// TIA Portal V19 export
DATA_BLOCK "A0302_PareggiatoreCoda_PERS"   // DB120
// stored: MemoryReserve 100
   VAR RETAIN
      Par : Struct
         Ax { S7_SetPoint := 'True'} : "Positioning_DOL_Machine_Par";
         Ax_Pers { ExternalAccessible := 'False'; ExternalVisible := 'False'; ExternalWritable := 'False'} : "Positioning_DOL_Machine_Pers_Data";
         Enc : "PosFbk_RTN";
         Ax_Aut { S7_SetPoint := 'True'} : "A0301_Mach_Speed_Par";
         Bloccaggio_Sens : Struct
            "2191B1" : "Analogic_SensorManagement_Par";
            SogliaWork { S7_SetPoint := 'True'} : Real := 0.0;
         END_STRUCT;
         CarroPareggCoda : Struct
            Delay_StartMove : Time := T#100MS;
            Preset { S7_SetPoint := 'True'} : LReal := 477.68;
         END_STRUCT;
         Cremaliera : Struct
            Modulo { S7_SetPoint := 'True'} : LReal := 2.5;
            Passo { S7_SetPoint := 'True'} : LReal := 7.854;
         END_STRUCT;
      END_STRUCT;
      Par_Sens : Struct
         AI { S7_SetPoint := 'True'} : "Analogic_SensorManagement_Par";
      END_STRUCT;
      Data_Sens { S7_SetPoint := 'True'} : "Analogic_SensorManagement_Data";
      Par_MachSens { S7_SetPoint := 'True'} : "A0301_Mach_Sens_Par";
      IEC_SP : Struct
         FTC_Input : Struct
            TON_PT : Time := T#10MS;
            TOF_PT : Time := T#100MS;
         END_STRUCT;
         FTC_Output : Struct
            TON_PT : Time := T#10MS;
            TOF_PT : Time := T#10MS;
         END_STRUCT;
         FTC_PresentMat : Struct
            TON_PT : Time := T#500MS;
            TOF_PT : Time := T#500MS;
         END_STRUCT;
         Check_2119B1 { ExternalAccessible := 'False'; ExternalVisible := 'False'; ExternalWritable := 'False'} : Struct
            TON_PT : Time := T#500MS;
         END_STRUCT;
      END_STRUCT;
   END_VAR
BEGIN
   Par.Ax.PosTolerance := 1.0;
   Par.Ax.Minus_Limit := 457.6;
   Par.Ax.Plus_Limit := 2845.0;
   Par.Ax.PreCutOff := 0.2;
   Par.Ax.PreEndLowSpeed := 2.0;
   Par.Ax.PreEndMedSpeed := 5.0;
   Par.Ax.LowSpeed := 2.0;
   Par.Ax.MedSpeed := 5.0;
   Par.Ax.HighSpeed := 50.0;
   Par.Ax.Man_Speed := 50.0;
   Par.Ax_Pers.AxisHomed := TRUE;
   Par.Enc.Preset.Pulses := 1_666_530_232;
   Par.Enc.Preset.Units := 477.68;
   Par.Enc.Config.Resolution := 125.663706143592;
   Par.Ax_Aut.SemiAut_Vel := 50.0;
   Par.Ax_Aut.Aut_Vel := 50.0;
   Par.Ax_Aut.Aut_Acc := 1.0;
   Par.Ax_Aut.Aut_Dec := 1.0;
   Par.Bloccaggio_Sens."2191B1".Enable := TRUE;
   Par.Bloccaggio_Sens."2191B1".RangeLow := 0.0;
   Par.Bloccaggio_Sens."2191B1".RangeHigh := 0.0;
   Par_Sens.AI.Enable := TRUE;
   Par_Sens.AI.RangeLow := 43.0;
   Par_Sens.AI.RangeHigh := 133.7;
   Data_Sens.OffsetValue := -4.04816818237305;
   Data_Sens.OffsetValid := TRUE;
   Par_MachSens.Tol_Work := 89.3;
   Par_MachSens.WorkTime_SensDisable := T#10MS;
END_DATA_BLOCK
